(* IEC 61131-3 sources: Industry-PLC-LLM/data/PLCBEAD_repo/PLCBEAD_PLCEmbed-main/PLC-BEAD/Source/GEB/CPOL, 1 file *)

(* ---- CPOL.ST ---- *)
TYPE oscat_complex :
  STRUCT
	re : REAL;
	im : REAL;
  END_STRUCT;
END_TYPE

FUNCTION_BLOCK CPOL_Block
	VAR_INPUT
		L :	REAL;
		A :	REAL;
	END_VAR

	VAR_OUTPUT
		CPOL :	oscat_complex;
	END_VAR

	CPOL.re := L * COS(A);
	CPOL.im := L * SIN(A);
END_FUNCTION_BLOCK

PROGRAM program0
  VAR
    LocalVar0 : REAL;
	LocalVaR1  : REAL;
	CPOL  : oscat_complex;
	func_block : CPOL_Block;
  END_VAR
	func_block.L  := LocalVar0;
	func_block.A  := LocalVaR1 ;
	func_block();
	CPOL := func_block.CPOL;
END_PROGRAM
